FUNCTION_BLOCK DieselMotor EXTENDS Motor

METHOD PUBLIC LoadFuel
ADSLOGSTR(    msgCtrlMask:=ADSLOG_MSGTYPE_LOG,
              msgFmtStr:='Loading fuel into the Diesel motor...',
              strArg:='');
END_METHOD

METHOD PUBLIC SpeedUp
ADSLOGSTR(    msgCtrlMask:=ADSLOG_MSGTYPE_LOG,
              msgFmtStr:='Accelerating the Diesel motor...',
              strArg:='');
END_METHOD

METHOD PUBLIC StartUp
ADSLOGSTR(    msgCtrlMask:=ADSLOG_MSGTYPE_LOG,
              msgFmtStr:='Starting the Diesel motor...',
              strArg:='');
END_METHOD

METHOD PUBLIC Stop
ADSLOGSTR(    msgCtrlMask:=ADSLOG_MSGTYPE_LOG,
              msgFmtStr:='Stopping the Diesel motor...',
              strArg:='');
END_METHOD

END_FUNCTION_BLOCK

(* stored: Version 1.1.0.1, ProductVersion 3.1.4024.12
   POU DieselMotor: Id {7cf974ad-c710-442b-a6a6-9485e8bb6eb3}, SpecialFunc None
   Method LoadFuel: Id {57b452c4-b864-4644-bedd-3268e3b336fe}
   Method SpeedUp: Id {d705be07-c977-442a-8dd2-753251f29f43}
   Method StartUp: Id {5be5d466-fbca-494b-8231-6205404a4c01}
   Method Stop: Id {da592090-4a88-4497-9996-23d0ab3145b4} *)
